Universal Robots PolyScope program: debugger_on_off_5s.urp

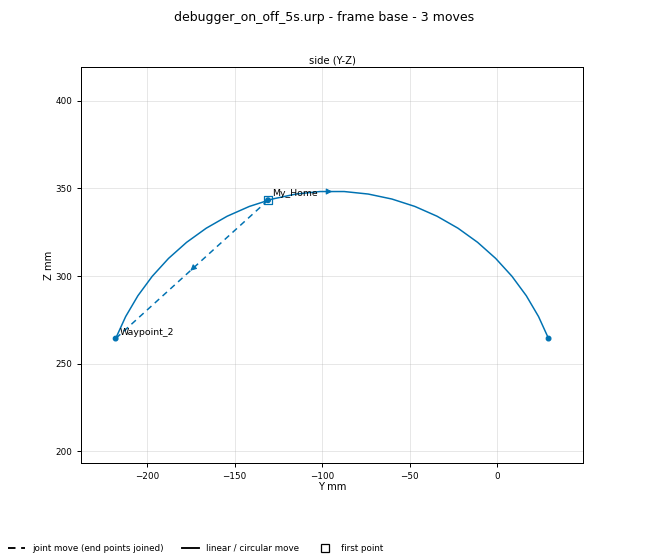
[picture p0: tool path of debugger_on_off_5s.urp in frame base, 3 of 4 moves have a stored position in this frame; points joined in program order, loops and branches not executed]
Program debugger_on_off_5s (installation=debugger_on_off_5s directory=/ursim/programs/new folder createdIn=5.21.0 lastSavedIn=5.21.0 robotSerialNumber=20195599999)
Calibrated DH parameters: a=[0, -0.425, -0.3922, 0, 0, 0]; d=[0.1625, 0, 0, 0.1333, 0.0997, 0.0996]; alpha=[1.570796, 0, 0, 1.570796, -1.570796, 0]; deltaTheta=[0, 0, 0, 0, 0, 0]
InitVariablesNode
Robot Program (runOnlyOnce=false)
  MoveJ speed 60 deg/s, acceleration 80 deg/s^2 (useActiveTCP=true optimoveEnabled=false optiMoveSpeed=0.3 optiMoveAcceleration=0.09) feature=Base
    Waypoint My_Home: TCP in base x=439.73 y=-130.88 z=343.272 mm, rx=2.2546 ry=-2.1864 rz=-0.0556 rad; joints [0, -86.876, -114.272, -70.325, 91.392, -1.776] deg
  Loop While (checkContinuously=false) expression=read_port_register(128)≟0
    Wait Sleep waitTime=0.5
  Script: write_port_register(128,0)
  MoveJ speed 60 deg/s, acceleration 80 deg/s^2 (useActiveTCP=true optimoveEnabled=false optiMoveSpeed=0.3 optiMoveAcceleration=0.09) feature=Base
    Waypoint Waypoint_2: TCP in base x=439.73 y=-217.891 z=264.28 mm, rx=2.2546 ry=-2.1864 rz=-0.0556 rad; joints [-10.828, -96.751, -116.976, -57.981, 91.091, -12.603] deg
  MoveP speed 250 mm/s, acceleration 1200 mm/s^2 (blendRadius=0.025 useActiveTCP=true optimoveEnabled=false optiMoveSpeed=0.3 optiMoveAcceleration=0.09) feature=Base
    CircleMove (OrientationMode=FIXED)
      Waypoint My_Home: TCP in base x=439.73 y=-130.88 z=343.272 mm, rx=2.2546 ry=-2.1864 rz=-0.0556 rad; joints [0, -86.876, -114.272, -70.325, 91.392, -1.776] deg
      Waypoint EndPoint_1: TCP in base x=439.73 y=29.293 z=264.28 mm, rx=2.2546 ry=-2.1864 rz=-0.0556 rad; joints [20.984, -89.956, -124.546, -56.375, 91.828, 19.212] deg
